# EPICS autosave request: BPMApp/Db/BPMSwitching_settings.req
$(P)$(R)SwMode-Sel
$(P)$(R)SwDeswapDly-SP
$(P)$(R)SwDivClk-SP
